// TwinCAT 3 PLC project MAS418_PLC2
// ProgramVersion: 3.1.4023.0
// libraries:
//   Tc2_Standard, * (Beckhoff Automation GmbH)
//   Tc2_System, * (Beckhoff Automation GmbH)
//   Tc3_Module, * (Beckhoff Automation GmbH)
// project tree:
//   / PlcTask.TcTTO
//   POUs/ MAIN.TcPOU
//   Task1/ GVL.TcGVL, POU.TcPOU
// real-time tasks:
//   TASK PlcTask: cycle T#10ms, priority 20, ADS port 350

CONFIGURATION MAS418_PLC2
    RESOURCE PLC ON TwinCAT3
        TASK PlcTask(INTERVAL := T#10ms, PRIORITY := 20);
        PROGRAM MAIN WITH PlcTask : MAIN;
    END_RESOURCE
END_CONFIGURATION

// ---- Task1/GVL.TcGVL
{attribute 'qualified_only'}
VAR_GLOBAL
	TimeDateInit : DATE_AND_TIME := DATE_AND_TIME#2023-2-7-14:51:0;
	TimeInit : TIME := TIME#5000MS;
END_VAR

// ---- POUs/MAIN.TcPOU
PROGRAM MAIN
VAR
END_VAR

POU();

END_PROGRAM

// ---- Task1/POU.TcPOU
PROGRAM POU
VAR
	pointer1 : POINTER TO DATE_AND_TIME := ADR(GVL.TimeDateInit);
	reference1 : REFERENCE TO TIME REF= GVL.TimeInit;
END_VAR

pointer1^ := DT#2024-2-8-14:51:0;
reference1 := TIME#4000ms;

END_PROGRAM
